// SIMATIC STEP 7 (V5.x) project linCC_test
// CPU: WinLC RTX
// station: P_ADR_BUS
// station: P_ADR_BUS
// station: Configurazione
// station: Stazione PC SIMATIC
// program: Programma S7(1)

SYMBOL_TABLE
"TankLevels"	DB 100	DB 100
"TankCtrl"	DB 200	DB 200
"cpuCycle"	MD 300	DWORD
"udtTankCtrl"	UDT 200	UDT 200
END_SYMBOL_TABLE

TYPE "udtTankCtrl"	// UDT 200
VERSION : 0.1
  STRUCT
   TankLoading : BOOL ;
   TankDischarging : BOOL ;
   TankLoad : BOOL ;
   TankDischarge : BOOL ;
   TankBusy : BOOL ;
   TankFull : BOOL ;
   TankEmpty : BOOL ;
  END_STRUCT ;	
END_TYPE

FUNCTION FC 10 : VOID
VERSION : 0.1
VAR_TEMP
  _bit1 : BOOL ;
  _500ms : BOOL ;
  _tempDI : DINT ;
END_VAR
BEGIN
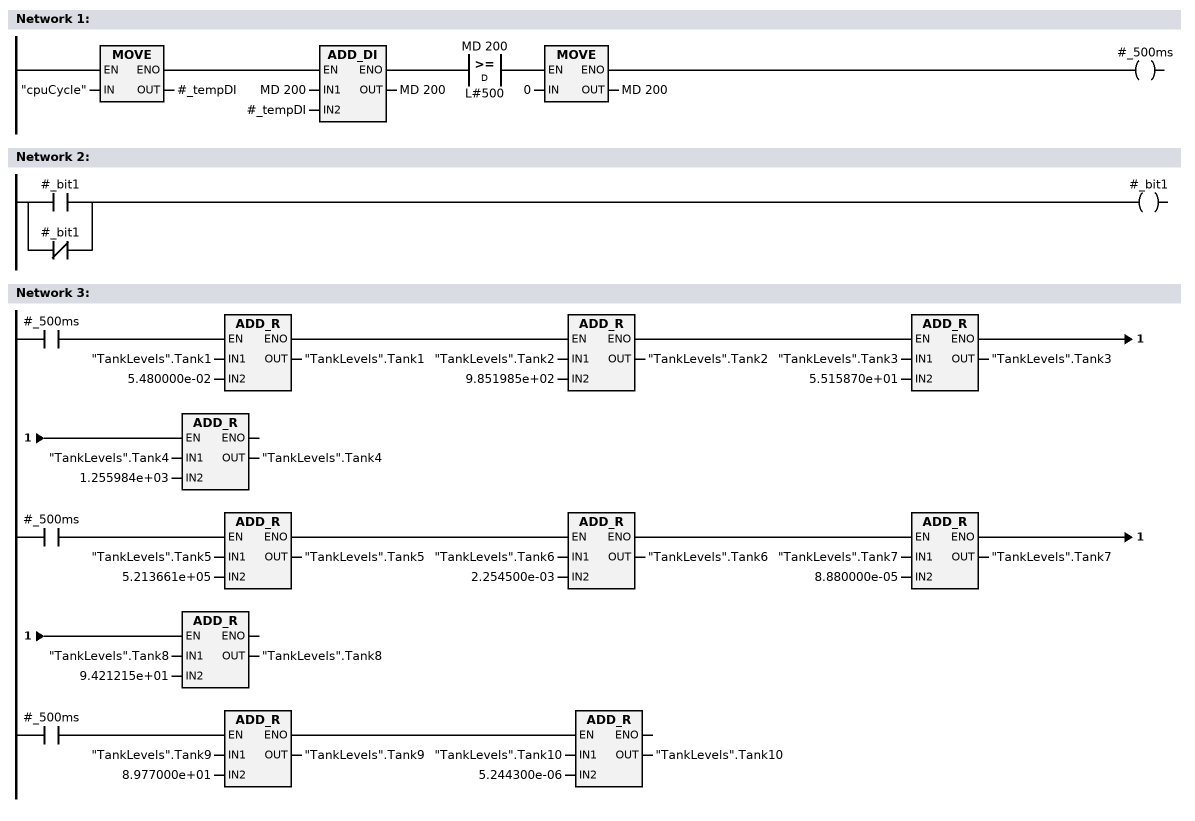
NETWORK
TITLE =
      A(;
      A(;
      L     "cpuCycle";
      T     #_tempDI;
      SET;
      SAVE;
      CLR;
      A     BR;
      );
      JNB   _001;
      L     MD 200;
      L     #_tempDI;
      +D;
      T     MD 200;
      AN    OV;
      SAVE;
      CLR;
_001: A     BR;
      );
      A(;
      L     MD 200;
      L     L#500;
      >=D;
      );
      JNB   _002;
      L     0;
      T     MD 200;
      SET;
      SAVE;
      CLR;
_002: A     BR;
      =     #_500ms;
NETWORK
TITLE =
      O     #_bit1;
      ON    #_bit1;
      =     #_bit1;
NETWORK
TITLE =
      A     #_500ms;
      =     L 6.0;
      A(;
      A(;
      A(;
      A     L 6.0;
      JNB   _003;
      L     "TankLevels".Tank1;
      L     5.480000e-02;
      +R;
      T     "TankLevels".Tank1;
      AN    OV;
      SAVE;
      CLR;
_003: A     BR;
      );
      JNB   _004;
      L     "TankLevels".Tank2;
      L     9.851985e+02;
      +R;
      T     "TankLevels".Tank2;
      AN    OV;
      SAVE;
      CLR;
_004: A     BR;
      );
      JNB   _005;
      L     "TankLevels".Tank3;
      L     5.515870e+01;
      +R;
      T     "TankLevels".Tank3;
      AN    OV;
      SAVE;
      CLR;
_005: A     BR;
      );
      JNB   _006;
      L     "TankLevels".Tank4;
      L     1.255984e+03;
      +R;
      T     "TankLevels".Tank4;
_006: NOP   0;
      A(;
      A(;
      A(;
      A     L 6.0;
      JNB   _007;
      L     "TankLevels".Tank5;
      L     5.213661e+05;
      +R;
      T     "TankLevels".Tank5;
      AN    OV;
      SAVE;
      CLR;
_007: A     BR;
      );
      JNB   _008;
      L     "TankLevels".Tank6;
      L     2.254500e-03;
      +R;
      T     "TankLevels".Tank6;
      AN    OV;
      SAVE;
      CLR;
_008: A     BR;
      );
      JNB   _009;
      L     "TankLevels".Tank7;
      L     8.880000e-05;
      +R;
      T     "TankLevels".Tank7;
      AN    OV;
      SAVE;
      CLR;
_009: A     BR;
      );
      JNB   _00a;
      L     "TankLevels".Tank8;
      L     9.421215e+01;
      +R;
      T     "TankLevels".Tank8;
_00a: NOP   0;
      A(;
      A     L 6.0;
      JNB   _00f;
      L     "TankLevels".Tank9;
      L     8.977000e+01;
      +R;
      T     "TankLevels".Tank9;
      AN    OV;
      SAVE;
      CLR;
_00f: A     BR;
      );
      JNB   _010;
      L     "TankLevels".Tank10;
      L     5.244300e-06;
      +R;
      T     "TankLevels".Tank10;
_010: NOP   0;
NETWORK
TITLE =
      A     #_bit1;
      =     L 6.0;
      A     L 6.0;
      A     "TankCtrl".Tank.TankLoad;
      =     "TankCtrl".Tank.TankLoading;
      A     L 6.0;
      A     "TankCtrl".Tank.TankDischarge;
      =     "TankCtrl".Tank.TankDischarging;
      A     L 6.0;
      A(;
      O     "TankCtrl".Tank.TankLoading;
      O     "TankCtrl".Tank.TankDischarging;
      O     "TankCtrl".Tank.TankFull;
      );
      =     "TankCtrl".Tank.TankBusy;
      A     L 6.0;
      A     #_500ms;
      =     L 6.1;
      A(;
      A     L 6.1;
      A     "TankCtrl".Tank.TankLoading;
      JNB   _011;
      L     "TankLevels".Tank1;
      L     1.000000e+01;
      +R;
      T     "TankLevels".Tank1;
      AN    OV;
      SAVE;
      CLR;
_011: A     BR;
      );
      A(;
      L     "TankLevels".Tank1;
      L     5.000000e+03;
      >=R;
      );
      JNB   _012;
      L     5.000000e+03;
      T     "TankLevels".Tank1;
_012: NOP   0;
      A(;
      A     L 6.1;
      A     "TankCtrl".Tank.TankDischarging;
      JNB   _013;
      L     "TankLevels".Tank1;
      L     1.000000e+01;
      -R;
      T     "TankLevels".Tank1;
      AN    OV;
      SAVE;
      CLR;
_013: A     BR;
      );
      A(;
      L     "TankLevels".Tank1;
      L     0.000000e+00;
      <=R;
      );
      JNB   _014;
      L     0.000000e+00;
      T     "TankLevels".Tank1;
_014: NOP   0;
      A     L 6.0;
      A(;
      L     "TankLevels".Tank1;
      L     1.000000e+01;
      <=R;
      );
      =     "TankCtrl".Tank.TankEmpty;
      A     L 6.0;
      A(;
      L     "TankLevels".Tank1;
      L     4.950000e+03;
      >=R;
      );
      =     "TankCtrl".Tank.TankFull;
END_FUNCTION

DATA_BLOCK "TankLevels"	// DB 100
VERSION : 0.1
  STRUCT
   Tank1 : REAL ;	//Tank1 Level
   Tank2 : REAL ;	//Tank2 Level
   Tank3 : REAL ;	//Tank3 Level
   Tank4 : REAL ;	//Tank4 Level
   Tank5 : REAL ;	//Tank5 Level
   Tank6 : REAL ;	//Tank6 Level
   Tank7 : REAL ;	//Tank7 Level
   Tank8 : REAL ;	//Tank8 Level
   Tank9 : REAL ;	//Tank9 Level
   Tank10 : REAL ;	//Tank10 Level
  END_STRUCT ;	
BEGIN
END_DATA_BLOCK

DATA_BLOCK "TankCtrl"	// DB 200
VERSION : 0.1
  STRUCT
   Tank : UDT 200;	//Ctrl Tank 1
   Tank2 : UDT 200;	//Ctrl Tank 2
   Tank3 : UDT 200;	//Ctrl Tank 3
   Tank4 : UDT 200;	//Ctrl Tank 4
   Tank5 : UDT 200;	//Ctrl Tank 5
   Tank6 : UDT 200;	//Ctrl Tank 6
   Tank7 : UDT 200;	//Ctrl Tank 7
   Tank8 : UDT 200;	//Ctrl Tank 8
   Tank9 : UDT 200;	//Ctrl Tank 9
   Tank10 : UDT 200;	//Ctrl Tank 10
  END_STRUCT ;	
BEGIN
END_DATA_BLOCK

ORGANIZATION_BLOCK OB 1
TITLE = "Main Program Sweep (Cycle)"
VERSION : 0.1
VAR_TEMP
  OB1_EV_CLASS : BYTE ;	//Bits 0-3 = 1 (Coming event), Bits 4-7 = 1 (Event class 1)
  OB1_SCAN_1 : BYTE ;	//1 (Cold restart scan 1 of OB 1), 3 (Scan 2-n of OB 1)
  OB1_PRIORITY : BYTE ;	//Priority of OB Execution
  OB1_OB_NUMBR : BYTE ;	//1 (Organization block 1, OB1)
  OB1_RESERVED_1 : BYTE ;	//Reserved for system
  OB1_RESERVED_2 : BYTE ;	//Reserved for system
  OB1_PREV_CYCLE : INT ;	//Cycle time of previous OB1 scan (milliseconds)
  OB1_MIN_CYCLE : INT ;	//Minimum cycle time of OB1 (milliseconds)
  OB1_MAX_CYCLE : INT ;	//Maximum cycle time of OB1 (milliseconds)
  OB1_DATE_TIME : DATE_AND_TIME ;	//Date and time OB1 started
END_VAR
BEGIN
NETWORK
TITLE =
      L     #OB1_PREV_CYCLE;
      T     "cpuCycle";
      CALL  FC 10;
END_ORGANIZATION_BLOCK
